PROGRAM confirmSecagem
VAR
	tempSeca: STRING;
	
END_VAR

//ESTE PROGRAMA TRANSFORMA O INPUT DO DIALOG EM TEMPO DE SECAGEM

tempSeca:= 'T#';
tempSeca:= concat(tempseca, TIME_TO_STRING(gvl_p.arrStatusEstufas[2].tempoSecagem));
tempSeca:= concat(tempseca, 'H');

GVL_p.arrStatusEstufas[2].tempoSecagem := STRING_TO_TIME(tempSeca);

END_PROGRAM

(* stored: Version 1.1.0.1, ProductVersion 3.1.4024.12
   POU confirmSecagem: Id {b06d3d4f-deb2-4292-8665-7d9fcf5eb2b6}, SpecialFunc None *)
